{attribute addProperty BoxType "KL2641-0001"}
{attribute addProperty Id "Manual_StateAT %I*BOOL000ReservedAT %I*BOOL000OutputAT %Q*BOOL000"}
{attribute addProperty CRC "3682416049"}
{attribute addProperty SizeInBites "0"}
{attribute addProperty SizeInBytes "0"}
TYPE Channel_DB7D35B1 :
STRUCT
	{attribute addProperty Name "Manual_State"}
	Manual_State AT %I* : BOOL;
	{attribute addProperty Name "Reserved"}
	Reserved AT %I* : BOOL;
	{attribute addProperty Name "Output"}
	Output AT %Q* : BOOL;
END_STRUCT
END_TYPE

(* stored: Version 1.2.0.0, ProductVersion 3.1.4024.9
   DUT Channel_DB7D35B1: Id {ccb8bc45-fc5e-4381-88e6-8fa075e5d3b4} *)
